// TIA Portal V21 export
VAR_GLOBAL   // PLC tag table "KAllAdditivo"
END_VAR
VAR_GLOBAL CONSTANT   // user constants
   KALLAdditivo_PortataPrincipaleTroppoBassa : Int := 1;   // La mandata principale è troppo alta per l'utenza comandanta
   KALLAdditivo_PortataPrincipaleTroppoAlta : Int := 2;   // La mandata principale è troppo basssa per l'utenza comandata
END_VAR
